// TIA Portal V21 export
TYPE "Std_eValveMode"
   STRUCT
      MA01_Directional_control_valve_functions { ExternalVisible := 'False'} : Int := 1;
      MA02_Proportional_directional_control_valve { ExternalVisible := 'False'} : Int := 2;
      MA03_Proportional_pressure_regulation { ExternalVisible := 'False'} : Int := 3;
      MA04_Modelbased_proportional_pressure_regulation { ExternalVisible := 'False'} : Int := 4;
      MA05_Supply_and_exhaust_air_flow_control { ExternalVisible := 'False'} : Int := 5;
      MA06_ECO_drive { ExternalVisible := 'False'} : Int := 6;
      MA07_Presetting_of_travel_time { ExternalVisible := 'False'} : Int := 7;
      MA08_Selectable_pressure_level_ECO { ExternalVisible := 'False'} : Int := 8;
      MA10_Flow_control { ExternalVisible := 'False'} : Int := 10;
      MA11_Soft_stop { ExternalVisible := 'False'} : Int := 11;
      MA12_Leakage_diagnostics { ExternalVisible := 'False'} : Int := 12;
      MA32_Positioning_and_Force { ExternalVisible := 'False'} : Int := 32;
      MA33_Positioning { ExternalVisible := 'False'} : Int := 33;
      VM60_TeachIn_run { ExternalVisible := 'False'} : Int := 60;
      VM61_Inactive { ExternalVisible := 'False'} : Int := 61;
      VM63_Transfermode { ExternalVisible := 'False'} : Int := 63;
   END_STRUCT;
END_TYPE
